FUNCTION_BLOCK ValueChangeDetector
VAR_INPUT
	Value			:	INT;
END_VAR
VAR_OUTPUT
	ValueChanged	:	BOOL;
END_VAR
VAR
	ValueCurrent	:	INT;
	ValueMem		:	INT;
	SetInit			:	BOOL := TRUE;
END_VAR

(*
Detect value change
*)

ValueCurrent := Value;

ValueChanged := ValueCurrent<>ValueMem;

ValueMem:=ValueCurrent;

// set once to changed on init cycle
// it allows to send data after power recycle 
IF SetInit THEN
	SetInit := FALSE;
	ValueChanged := TRUE;
END_IF

END_FUNCTION_BLOCK

(* stored: Version 1.1.0.1, ProductVersion 3.1.4024.15
   POU ValueChangeDetector: Id {0a2548e8-235c-4d33-a26a-b06c3223e6ce}, SpecialFunc None *)
